(* CoDeSys 2.3.9.41 project: Разработка блока управления конвейерной системы [тележка].pro *)
(* Libraries: Standard.lib 4.10.05 11:14:46, IecSfc.lib 13.4.06 15:51:28, SYSLIBCALLBACK.LIB 26.9.08 16:43:52 *)

(* Global variable list: Global_Variables *)
VAR_GLOBAL
	Observer: BOOL;
	Warning: BOOL;
	Stop: BOOL;
	Start: BOOL;
END_VAR

(* POU PLC_PRG, FBD *)
PROGRAM PLC_PRG
VAR
	Trig1: R_TRIG;
	Trip2: F_TRIG;
	Timer1: TOF;
	Timer2: TON;
END_VAR
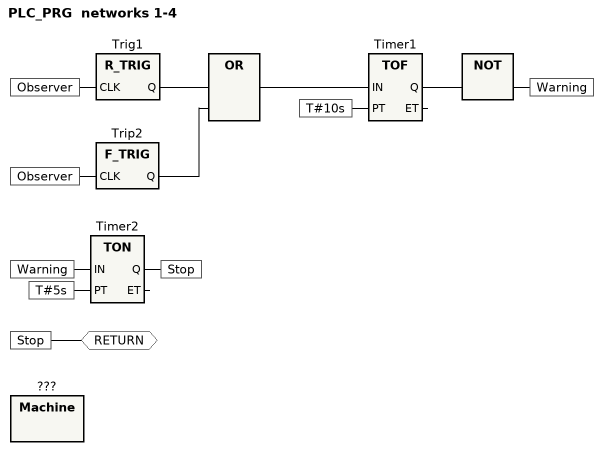
_FBD_ (* Function Block Diagram *)
NETWORK 1
	NOT Timer1:TOF(IN: OR(Trig1:R_TRIG(CLK: Observer), Trip2:F_TRIG(CLK: Observer)), PT: T#10s) => Warning
NETWORK 2
	Timer2:TON(IN: Warning, PT: T#5s) => Stop
NETWORK 3
	Stop => <RETURN>
NETWORK 4
	???:Machine()
_END_FBD_
END_PROGRAM

(* POU Machine, SFC *)
PROGRAM Machine
VAR
	X_pos: INT;
	Y_pos: INT;
	Counter: INT;
END_VAR
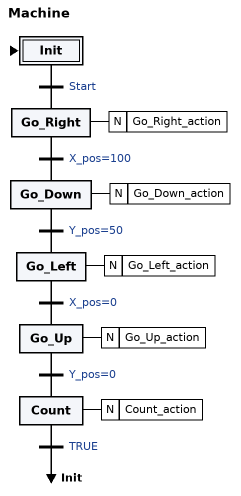
INITIAL_STEP Init:
END_STEP
TRANSITION FROM Init TO Go_Right := Start;
END_TRANSITION
STEP Go_Right:
	Go_Right_action(N);
END_STEP
TRANSITION FROM Go_Right TO Go_Down := X_pos=100;
END_TRANSITION
STEP Go_Down:
	Go_Down_action(N);
END_STEP
TRANSITION FROM Go_Down TO Go_Left := Y_pos=50;
END_TRANSITION
STEP Go_Left:
	Go_Left_action(N);
END_STEP
TRANSITION FROM Go_Left TO Go_Up := X_pos=0;
END_TRANSITION
STEP Go_Up:
	Go_Up_action(N);
END_STEP
TRANSITION FROM Go_Up TO Count := Y_pos=0;
END_TRANSITION
STEP Count:
	Count_action(N);
END_STEP
TRANSITION FROM Count TO Init := TRUE;
END_TRANSITION

ACTION Go_Right_action:
X_pos:=X_pos+1;
END_ACTION

ACTION Go_Down_action:
Y_pos:=Y_pos+1;
END_ACTION

ACTION Go_Left_action:
X_pos:=X_pos-1;
END_ACTION

ACTION Go_Up_action:
Y_pos:=Y_pos-1;
END_ACTION

ACTION Count_action:
Counter:=Counter+1;
END_ACTION
END_PROGRAM

(* Visualisation Observation
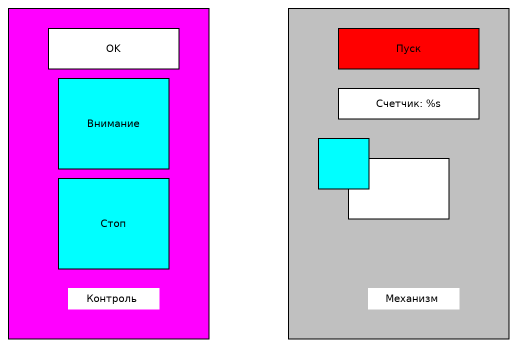
rectangle at (120,300)-(211,321): text "Контроль"
rectangle at (100,40)-(231,81): text "OK"; alarm colour if .Observer; taps .Observer
rounded rectangle at (110,90)-(221,181): text "Внимание"; alarm colour if .Warning
rounded rectangle at (110,190)-(221,281): text "Стоп"; alarm colour if .Stop
rectangle at (390,40)-(531,81): text "Пуск"; alarm colour if .Start; taps .Start
rectangle at (390,100)-(531,131): text "Счетчик: %s"; shows Machine.Counter
rectangle at (370,150)-(421,201): x offset Machine.X_pos; y offset Machine.Y_pos
rectangle at (420,300)-(511,321): text "Механизм"
3 more shapes without text or variables
*)
